INTERFACE I_Symbol EXTENDS I_GraphicalElement

PROPERTY PUBLIC FlipX : BOOL
GET
END_GET
SET
END_SET
END_PROPERTY

PROPERTY PUBLIC FlipY : BOOL
GET
END_GET
SET
END_SET
END_PROPERTY

PROPERTY PUBLIC Rotation : UINT
GET
END_GET
SET
END_SET
END_PROPERTY

END_INTERFACE

(* stored: Version 1.1.0.1, ProductVersion 3.1.4024.15
   Itf I_Symbol: Id {6e35cf10-53ed-0be2-099e-ea627d0ab8f6}
   Property FlipX: Id {3c4357a1-63f5-0772-1123-93e77bd8fdd7}
   Get Get: Id {b89aa9af-5325-0af6-2b86-23b7c1be5a36}
   Set Set: Id {6be0f5d4-0854-07b5-2c64-59e52360e520}
   Property FlipY: Id {e9419acc-fcd4-0fd8-3467-c66e002bee65}
   Get Get: Id {9de9ef6a-b96b-0612-3039-072bf8ad3054}
   Set Set: Id {b53bcc6f-41ee-0852-2069-6701ba4e176b}
   Property Rotation: Id {93721753-6e82-0a12-0905-8298f9167ad9}
   Get Get: Id {a12fde2b-ccea-0f93-25b9-6e8520b9db6c}
   Set Set: Id {6e336aa8-4877-09cc-002a-ac0f1cb7ff4b} *)
